// TIA Portal V17 export
// export: Created 2022-12-09T10:51:17.0895066Z, ExportSetting WithDefaults, DisplayName Totally Integrated Automation Portal, DisplayVersion V17 Update 5, DisplayName TIA Portal Openness, DisplayVersion V17 Update 5, DisplayName TIA Portal Version Control Interface, DisplayVersion V17, DisplayName Simotion SCOUT TIA, DisplayVersion 5.4.3.0, DisplayName SINAMICS Startdrive Advanced, DisplayVersion V17 SP1, DisplayName SINAMICS Startdrive G130, G150, S120, S150, SINAMICS MV, S210, DisplayVersion V17 SP1, DisplayName SINAMICS Startdrive G110M, G120, G120C, G120D, G120P, G115D, DisplayVersion V17 SP1, DisplayName STEP 7 Professional, DisplayVersion V17 Update 5, DisplayName STEP 7 Safety, DisplayVersion V17, DisplayName WinCC Advanced, DisplayVersion V17 Update 5
TYPE "NDSN_ST_ADIList"
// stored: IsFailsafeCompliant false
   STRUCT
      NDSN_ST_ADI_List { S7_SetPoint := 'True'} : Array[0..49] of "NDSN_ST_ADI";
   END_STRUCT;
   // NDSN_ST_ADI_List[0].i_ADI := 11682;
   // NDSN_ST_ADI_List[1].i_ADI := 11683;
   // NDSN_ST_ADI_List[2].i_ADI := 10853;
   // NDSN_ST_ADI_List[3].i_ADI := 10855;
   // NDSN_ST_ADI_List[4].i_ADI := 10858;
   // NDSN_ST_ADI_List[5].i_ADI := 10859;
   // NDSN_ST_ADI_List[6].i_ADI := 10860;
   // NDSN_ST_ADI_List[7].i_ADI := 11376;
   // NDSN_ST_ADI_List[8].i_ADI := 11378;
   // NDSN_ST_ADI_List[9].i_ADI := 10002;
   // NDSN_ST_ADI_List[10].i_ADI := 10547;
   // NDSN_ST_ADI_List[11].i_ADI := 10549;
   // NDSN_ST_ADI_List[12].i_ADI := 10548;
   // NDSN_ST_ADI_List[13].i_ADI := 6203;
   // NDSN_ST_ADI_List[14].i_ADI := 6102;
   // NDSN_ST_ADI_List[15].i_ADI := 6946;
   // NDSN_ST_ADI_List[16].i_ADI := 7046;
   // NDSN_ST_ADI_List[17].i_ADI := 7146;
   // NDSN_ST_ADI_List[18].i_ADI := 7147;
   // NDSN_ST_ADI_List[19].i_ADI := 7148;
   // NDSN_ST_ADI_List[20].i_ADI := 7248;
   // NDSN_ST_ADI_List[21].i_ADI := 13017;
   // NDSN_ST_ADI_List[22].i_ADI := 13003;
   // NDSN_ST_ADI_List[23].i_ADI := 13008;
   // NDSN_ST_ADI_List[24].i_ADI := 13009;
   // NDSN_ST_ADI_List[25].i_ADI := 13012;
   // NDSN_ST_ADI_List[26].i_ADI := 801;
   // NDSN_ST_ADI_List[27].i_ADI := 19;
   // NDSN_ST_ADI_List[28].i_ADI := 22;
   // NDSN_ST_ADI_List[29].i_ADI := 11681;
   // NDSN_ST_ADI_List[30].i_ADI := 11685;
   // NDSN_ST_ADI_List[31].i_ADI := 6103;
   // NDSN_ST_ADI_List[32].i_ADI := 6002;
   // NDSN_ST_ADI_List[33].i_ADI := 13002;
   // NDSN_ST_ADI_List[34].i_ADI := 13;
   // NDSN_ST_ADI_List[35].i_ADI := 16;
   // NDSN_ST_ADI_List[36].i_ADI := 29;
   // NDSN_ST_ADI_List[37].i_ADI := 30;
   // NDSN_ST_ADI_List[0..1].i_Size := 36;
   // NDSN_ST_ADI_List[2..12].i_Size := 2;
   // NDSN_ST_ADI_List[13].i_Size := 4;
   // NDSN_ST_ADI_List[14].i_Size := 2;
   // NDSN_ST_ADI_List[15..16].i_Size := 4;
   // NDSN_ST_ADI_List[17..18].i_Size := 2;
   // NDSN_ST_ADI_List[19..20].i_Size := 4;
   // NDSN_ST_ADI_List[21..28].i_Size := 2;
   // NDSN_ST_ADI_List[29..30].i_Size := 36;
   // NDSN_ST_ADI_List[31].i_Size := 4;
   // NDSN_ST_ADI_List[32..34].i_Size := 2;
   // NDSN_ST_ADI_List[35].i_Size := 4;
   // NDSN_ST_ADI_List[36].i_Size := 2;
   // NDSN_ST_ADI_List[37].i_Size := 8;
END_TYPE
